// TIA Portal V17 export
// export: Created 2024-08-26T21:10:52.0065134Z, ExportSetting WithDefaults, DisplayName Totally Integrated Automation Portal, DisplayVersion V17 Update 7, DisplayName TIA Portal Openness, DisplayVersion V17 Update 7, DisplayName TIA Portal Version Control Interface, DisplayVersion V17, DisplayName SINAMICS Startdrive Advanced, DisplayVersion V17 SP2, DisplayName SINAMICS Startdrive G110M, G120, G120C, G120D, G120P, G115D, DisplayVersion V17 SP2, DisplayName SINAMICS Startdrive G130, G150, S120, S150, SINAMICS MV, S210, DisplayVersion V17 SP2, DisplayName STEP 7 Professional, DisplayVersion V17 Update 7, DisplayName STEP 7 Safety, DisplayVersion V17 Update 6, DisplayName WinCC Advanced / Unified PC, DisplayVersion V17 Update 7
DATA_BLOCK "DB_MAIN_IJCORE"   // DB1000
{ S7_Optimized_Access := 'FALSE' }
VERSION : 0.1
// stored: AutoNumber false, DBAccessibleFromOPCUA true, DBAccessibleFromWebserver true, IsOnlyStoredInLoadMemory false, IsWriteProtectedInAS false
   VAR
      Enable : Bool := true;   // Enable traceability
      Mode : USInt := 1;   // 1. Full traceability, 2. Downgrade Mode
      Errors : Word;   // Error code
      hmiInd : USInt;   // Global Indicator Status
      CreatedNFP : Array[1.."MaxCreateNFP"] of String[30];   // Created NFP
      STAT : Struct
         STA_OK : Bool;
         PFC_OK : Bool;
         TRC_OK : Bool;
         CNF_OK : Bool;
         TRR_OK : Bool;
         ProcessResults : USInt;   // 1: Part OK, 2: PartNOK
      END_STRUCT;
      CMD : Struct
         STA : Bool;
         PFC : Bool;
         TRC : Bool;
         CNF : Bool;
         TRR : Bool;
      END_STRUCT;
   END_VAR
BEGIN
END_DATA_BLOCK
